        FuUnicodeCodepointCaseConvert := 66571;
        RETURN;
    66612:
        FuUnicodeCodepointCaseConvert := 66572;
        RETURN;
    66613:
        FuUnicodeCodepointCaseConvert := 66573;
        RETURN;
    66614:
        FuUnicodeCodepointCaseConvert := 66574;
        RETURN;
    66615:
        FuUnicodeCodepointCaseConvert := 66575;
        RETURN;
    66616:
        FuUnicodeCodepointCaseConvert := 66576;
        RETURN;
    66617:
        FuUnicodeCodepointCaseConvert := 66577;
        RETURN;
    66618:
        FuUnicodeCodepointCaseConvert := 66578;
        RETURN;
    66619:
        FuUnicodeCodepointCaseConvert := 66579;
        RETURN;
    66620:
        FuUnicodeCodepointCaseConvert := 66580;
        RETURN;
    66621:
        FuUnicodeCodepointCaseConvert := 66581;
        RETURN;
    66622:
        FuUnicodeCodepointCaseConvert := 66582;
        RETURN;
    66623:
        FuUnicodeCodepointCaseConvert := 66583;
        RETURN;
    66624:
        FuUnicodeCodepointCaseConvert := 66584;
        RETURN;
    66625:
        FuUnicodeCodepointCaseConvert := 66585;
        RETURN;
    66626:
        FuUnicodeCodepointCaseConvert := 66586;
        RETURN;
    66627:
        FuUnicodeCodepointCaseConvert := 66587;
        RETURN;
    66628:
        FuUnicodeCodepointCaseConvert := 66588;
        RETURN;
    66629:
        FuUnicodeCodepointCaseConvert := 66589;
        RETURN;
    66630:
        FuUnicodeCodepointCaseConvert := 66590;
        RETURN;
    66631:
        FuUnicodeCodepointCaseConvert := 66591;
        RETURN;
    66632:
        FuUnicodeCodepointCaseConvert := 66592;
        RETURN;
    66633:
        FuUnicodeCodepointCaseConvert := 66593;
        RETURN;
    66634:
        FuUnicodeCodepointCaseConvert := 66594;
        RETURN;
    66635:
        FuUnicodeCodepointCaseConvert := 66595;
        RETURN;
    66636:
        FuUnicodeCodepointCaseConvert := 66596;
        RETURN;
    66637:
        FuUnicodeCodepointCaseConvert := 66597;
        RETURN;
    66638:
        FuUnicodeCodepointCaseConvert := 66598;
        RETURN;
    66639:
        FuUnicodeCodepointCaseConvert := 66599;
        RETURN;
    66736:
        FuUnicodeCodepointCaseConvert := 66776;
        RETURN;
    66737:
        FuUnicodeCodepointCaseConvert := 66777;
        RETURN;
    66738:
        FuUnicodeCodepointCaseConvert := 66778;
        RETURN;
    66739:
        FuUnicodeCodepointCaseConvert := 66779;
        RETURN;
    66740:
        FuUnicodeCodepointCaseConvert := 66780;
        RETURN;
    66741:
        FuUnicodeCodepointCaseConvert := 66781;
        RETURN;
    66742:
        FuUnicodeCodepointCaseConvert := 66782;
        RETURN;
    66743:
        FuUnicodeCodepointCaseConvert := 66783;
        RETURN;
    66744:
        FuUnicodeCodepointCaseConvert := 66784;
        RETURN;
    66745:
        FuUnicodeCodepointCaseConvert := 66785;
        RETURN;
    66746:
        FuUnicodeCodepointCaseConvert := 66786;
        RETURN;
    66747:
        FuUnicodeCodepointCaseConvert := 66787;
        RETURN;
    66748:
        FuUnicodeCodepointCaseConvert := 66788;
        RETURN;
    66749:
        FuUnicodeCodepointCaseConvert := 66789;
        RETURN;
    66750:
        FuUnicodeCodepointCaseConvert := 66790;
        RETURN;
    66751:
        FuUnicodeCodepointCaseConvert := 66791;
        RETURN;
    66752:
        FuUnicodeCodepointCaseConvert := 66792;
        RETURN;
    66753:
        FuUnicodeCodepointCaseConvert := 66793;
        RETURN;
    66754:
        FuUnicodeCodepointCaseConvert := 66794;
        RETURN;
    66755:
        FuUnicodeCodepointCaseConvert := 66795;
        RETURN;
    66756:
        FuUnicodeCodepointCaseConvert := 66796;
        RETURN;
    66757:
        FuUnicodeCodepointCaseConvert := 66797;
        RETURN;
    66758:
        FuUnicodeCodepointCaseConvert := 66798;
        RETURN;
    66759:
        FuUnicodeCodepointCaseConvert := 66799;
        RETURN;
    66760:
        FuUnicodeCodepointCaseConvert := 66800;
        RETURN;
    66761:
        FuUnicodeCodepointCaseConvert := 66801;
        RETURN;
    66762:
        FuUnicodeCodepointCaseConvert := 66802;
        RETURN;
    66763:
        FuUnicodeCodepointCaseConvert := 66803;
        RETURN;
    66764:
        FuUnicodeCodepointCaseConvert := 66804;
        RETURN;
    66765:
        FuUnicodeCodepointCaseConvert := 66805;
        RETURN;
    66766:
        FuUnicodeCodepointCaseConvert := 66806;
        RETURN;
    66767:
        FuUnicodeCodepointCaseConvert := 66807;
        RETURN;
    66768:
        FuUnicodeCodepointCaseConvert := 66808;
        RETURN;
    66769:
        FuUnicodeCodepointCaseConvert := 66809;
        RETURN;
    66770:
        FuUnicodeCodepointCaseConvert := 66810;
        RETURN;
    66771:
        FuUnicodeCodepointCaseConvert := 66811;
        RETURN;
    66776:
        FuUnicodeCodepointCaseConvert := 66736;
        RETURN;
    66777:
        FuUnicodeCodepointCaseConvert := 66737;
        RETURN;
    66778:
        FuUnicodeCodepointCaseConvert := 66738;
        RETURN;
    66779:
        FuUnicodeCodepointCaseConvert := 66739;
        RETURN;
    66780:
        FuUnicodeCodepointCaseConvert := 66740;
        RETURN;
    66781:
        FuUnicodeCodepointCaseConvert := 66741;
        RETURN;
    66782:
        FuUnicodeCodepointCaseConvert := 66742;
        RETURN;
    66783:
        FuUnicodeCodepointCaseConvert := 66743;
        RETURN;
    66784:
        FuUnicodeCodepointCaseConvert := 66744;
        RETURN;
    66785:
        FuUnicodeCodepointCaseConvert := 66745;
        RETURN;
    66786:
        FuUnicodeCodepointCaseConvert := 66746;
        RETURN;
    66787:
        FuUnicodeCodepointCaseConvert := 66747;
        RETURN;
    66788:
        FuUnicodeCodepointCaseConvert := 66748;
        RETURN;
    66789:
        FuUnicodeCodepointCaseConvert := 66749;
        RETURN;
    66790:
        FuUnicodeCodepointCaseConvert := 66750;
        RETURN;
    66791:
        FuUnicodeCodepointCaseConvert := 66751;
        RETURN;
    66792:
        FuUnicodeCodepointCaseConvert := 66752;
        RETURN;
    66793:
        FuUnicodeCodepointCaseConvert := 66753;
        RETURN;
    66794:
        FuUnicodeCodepointCaseConvert := 66754;
        RETURN;
    66795:
        FuUnicodeCodepointCaseConvert := 66755;
        RETURN;
    66796:
        FuUnicodeCodepointCaseConvert := 66756;
        RETURN;
    66797:
        FuUnicodeCodepointCaseConvert := 66757;
        RETURN;
    66798:
        FuUnicodeCodepointCaseConvert := 66758;
        RETURN;
    66799:
        FuUnicodeCodepointCaseConvert := 66759;
        RETURN;
    66800:
        FuUnicodeCodepointCaseConvert := 66760;
        RETURN;
    66801:
        FuUnicodeCodepointCaseConvert := 66761;
        RETURN;
    66802:
        FuUnicodeCodepointCaseConvert := 66762;
        RETURN;
    66803:
        FuUnicodeCodepointCaseConvert := 66763;
        RETURN;
    66804:
        FuUnicodeCodepointCaseConvert := 66764;
        RETURN;
    66805:
        FuUnicodeCodepointCaseConvert := 66765;
        RETURN;
    66806:
        FuUnicodeCodepointCaseConvert := 66766;
        RETURN;
    66807:
        FuUnicodeCodepointCaseConvert := 66767;
        RETURN;
    66808:
        FuUnicodeCodepointCaseConvert := 66768;
        RETURN;
    66809:
        FuUnicodeCodepointCaseConvert := 66769;
        RETURN;
    66810:
        FuUnicodeCodepointCaseConvert := 66770;
        RETURN;
    66811:
        FuUnicodeCodepointCaseConvert := 66771;
        RETURN;
    66928:
        FuUnicodeCodepointCaseConvert := 66967;
        RETURN;
    66929:
        FuUnicodeCodepointCaseConvert := 66968;
        RETURN;
    66930:
        FuUnicodeCodepointCaseConvert := 66969;
        RETURN;
    66931:
        FuUnicodeCodepointCaseConvert := 66970;
        RETURN;
    66932:
        FuUnicodeCodepointCaseConvert := 66971;
        RETURN;
    66933:
        FuUnicodeCodepointCaseConvert := 66972;
        RETURN;
    66934:
        FuUnicodeCodepointCaseConvert := 66973;
        RETURN;
    66935:
        FuUnicodeCodepointCaseConvert := 66974;
        RETURN;
    66936:
        FuUnicodeCodepointCaseConvert := 66975;
        RETURN;
    66937:
        FuUnicodeCodepointCaseConvert := 66976;
        RETURN;
    66938:
        FuUnicodeCodepointCaseConvert := 66977;
        RETURN;
    66940:
        FuUnicodeCodepointCaseConvert := 66979;
        RETURN;
    66941:
        FuUnicodeCodepointCaseConvert := 66980;
        RETURN;
    66942:
        FuUnicodeCodepointCaseConvert := 66981;
        RETURN;
    66943:
        FuUnicodeCodepointCaseConvert := 66982;
        RETURN;
    66944:
        FuUnicodeCodepointCaseConvert := 66983;
        RETURN;
    66945:
        FuUnicodeCodepointCaseConvert := 66984;
        RETURN;
    66946:
        FuUnicodeCodepointCaseConvert := 66985;
        RETURN;
    66947:
        FuUnicodeCodepointCaseConvert := 66986;
        RETURN;
    66948:
        FuUnicodeCodepointCaseConvert := 66987;
        RETURN;
    66949:
        FuUnicodeCodepointCaseConvert := 66988;
        RETURN;
    66950:
        FuUnicodeCodepointCaseConvert := 66989;
        RETURN;
    66951:
        FuUnicodeCodepointCaseConvert := 66990;
        RETURN;
    66952:
        FuUnicodeCodepointCaseConvert := 66991;
        RETURN;
    66953:
        FuUnicodeCodepointCaseConvert := 66992;
        RETURN;
    66954:
        FuUnicodeCodepointCaseConvert := 66993;
        RETURN;
    66956:
        FuUnicodeCodepointCaseConvert := 66995;
        RETURN;
    66957:
        FuUnicodeCodepointCaseConvert := 66996;
        RETURN;
    66958:
        FuUnicodeCodepointCaseConvert := 66997;
        RETURN;
    66959:
        FuUnicodeCodepointCaseConvert := 66998;
        RETURN;
    66960:
        FuUnicodeCodepointCaseConvert := 66999;
        RETURN;
    66961:
        FuUnicodeCodepointCaseConvert := 67000;
        RETURN;
    66962:
        FuUnicodeCodepointCaseConvert := 67001;
        RETURN;
    66964:
        FuUnicodeCodepointCaseConvert := 67003;
        RETURN;
    66965:
        FuUnicodeCodepointCaseConvert := 67004;
        RETURN;
    66967:
        FuUnicodeCodepointCaseConvert := 66928;
        RETURN;
    66968:
        FuUnicodeCodepointCaseConvert := 66929;
        RETURN;
    66969:
        FuUnicodeCodepointCaseConvert := 66930;
        RETURN;
    66970:
        FuUnicodeCodepointCaseConvert := 66931;
        RETURN;
    66971:
        FuUnicodeCodepointCaseConvert := 66932;
        RETURN;
    66972:
        FuUnicodeCodepointCaseConvert := 66933;
        RETURN;
    66973:
        FuUnicodeCodepointCaseConvert := 66934;
        RETURN;
    66974:
        FuUnicodeCodepointCaseConvert := 66935;
        RETURN;
    66975:
        FuUnicodeCodepointCaseConvert := 66936;
        RETURN;
    66976:
        FuUnicodeCodepointCaseConvert := 66937;
        RETURN;
    66977:
        FuUnicodeCodepointCaseConvert := 66938;
        RETURN;
    66979:
        FuUnicodeCodepointCaseConvert := 66940;
        RETURN;
    66980:
        FuUnicodeCodepointCaseConvert := 66941;
        RETURN;
    66981:
        FuUnicodeCodepointCaseConvert := 66942;
        RETURN;
    66982:
        FuUnicodeCodepointCaseConvert := 66943;
        RETURN;
    66983:
        FuUnicodeCodepointCaseConvert := 66944;
        RETURN;
    66984:
        FuUnicodeCodepointCaseConvert := 66945;
        RETURN;
    66985:
        FuUnicodeCodepointCaseConvert := 66946;
        RETURN;
    66986:
        FuUnicodeCodepointCaseConvert := 66947;
        RETURN;
    66987:
        FuUnicodeCodepointCaseConvert := 66948;
        RETURN;
    66988:
        FuUnicodeCodepointCaseConvert := 66949;
        RETURN;
    66989:
        FuUnicodeCodepointCaseConvert := 66950;
        RETURN;
    66990:
        FuUnicodeCodepointCaseConvert := 66951;
        RETURN;
    66991:
        FuUnicodeCodepointCaseConvert := 66952;
        RETURN;
    66992:
        FuUnicodeCodepointCaseConvert := 66953;
        RETURN;
    66993:
        FuUnicodeCodepointCaseConvert := 66954;
        RETURN;
    66995:
        FuUnicodeCodepointCaseConvert := 66956;
        RETURN;
    66996:
        FuUnicodeCodepointCaseConvert := 66957;
        RETURN;
    66997:
        FuUnicodeCodepointCaseConvert := 66958;
        RETURN;
    66998:
        FuUnicodeCodepointCaseConvert := 66959;
        RETURN;
    66999:
        FuUnicodeCodepointCaseConvert := 66960;
        RETURN;
    67000:
        FuUnicodeCodepointCaseConvert := 66961;
        RETURN;
    67001:
        FuUnicodeCodepointCaseConvert := 66962;
        RETURN;
    67003:
        FuUnicodeCodepointCaseConvert := 66964;
        RETURN;
    67004:
        FuUnicodeCodepointCaseConvert := 66965;
        RETURN;
    68736:
        FuUnicodeCodepointCaseConvert := 68800;
        RETURN;
    68737:
        FuUnicodeCodepointCaseConvert := 68801;
        RETURN;
    68738:
        FuUnicodeCodepointCaseConvert := 68802;
        RETURN;
    68739:
        FuUnicodeCodepointCaseConvert := 68803;
        RETURN;
    68740:
        FuUnicodeCodepointCaseConvert := 68804;
        RETURN;
    68741:
        FuUnicodeCodepointCaseConvert := 68805;
        RETURN;
    68742:
        FuUnicodeCodepointCaseConvert := 68806;
        RETURN;
    68743:
        FuUnicodeCodepointCaseConvert := 68807;
        RETURN;
    68744:
        FuUnicodeCodepointCaseConvert := 68808;
        RETURN;
    68745:
        FuUnicodeCodepointCaseConvert := 68809;
        RETURN;
    68746:
        FuUnicodeCodepointCaseConvert := 68810;
        RETURN;
    68747:
        FuUnicodeCodepointCaseConvert := 68811;
        RETURN;
    68748:
        FuUnicodeCodepointCaseConvert := 68812;
        RETURN;
    68749:
        FuUnicodeCodepointCaseConvert := 68813;
        RETURN;
    68750:
        FuUnicodeCodepointCaseConvert := 68814;
        RETURN;
    68751:
        FuUnicodeCodepointCaseConvert := 68815;
        RETURN;
    68752:
        FuUnicodeCodepointCaseConvert := 68816;
        RETURN;
    68753:
        FuUnicodeCodepointCaseConvert := 68817;
        RETURN;
    68754:
        FuUnicodeCodepointCaseConvert := 68818;
        RETURN;
    68755:
        FuUnicodeCodepointCaseConvert := 68819;
        RETURN;
    68756:
        FuUnicodeCodepointCaseConvert := 68820;
        RETURN;
    68757:
        FuUnicodeCodepointCaseConvert := 68821;
        RETURN;
    68758:
        FuUnicodeCodepointCaseConvert := 68822;
        RETURN;
    68759:
        FuUnicodeCodepointCaseConvert := 68823;
        RETURN;
    68760:
        FuUnicodeCodepointCaseConvert := 68824;
        RETURN;
    68761:
        FuUnicodeCodepointCaseConvert := 68825;
        RETURN;
    68762:
        FuUnicodeCodepointCaseConvert := 68826;
        RETURN;
    68763:
        FuUnicodeCodepointCaseConvert := 68827;
        RETURN;
    68764:
        FuUnicodeCodepointCaseConvert := 68828;
        RETURN;
    68765:
        FuUnicodeCodepointCaseConvert := 68829;
        RETURN;
    68766:
        FuUnicodeCodepointCaseConvert := 68830;
        RETURN;
    68767:
        FuUnicodeCodepointCaseConvert := 68831;
        RETURN;
    68768:
        FuUnicodeCodepointCaseConvert := 68832;
        RETURN;
    68769:
        FuUnicodeCodepointCaseConvert := 68833;
        RETURN;
    68770:
        FuUnicodeCodepointCaseConvert := 68834;
        RETURN;
    68771:
        FuUnicodeCodepointCaseConvert := 68835;
        RETURN;
    68772:
        FuUnicodeCodepointCaseConvert := 68836;
        RETURN;
    68773:
        FuUnicodeCodepointCaseConvert := 68837;
        RETURN;
    68774:
        FuUnicodeCodepointCaseConvert := 68838;
        RETURN;
    68775:
        FuUnicodeCodepointCaseConvert := 68839;
        RETURN;
    68776:
        FuUnicodeCodepointCaseConvert := 68840;
        RETURN;
    68777:
        FuUnicodeCodepointCaseConvert := 68841;
        RETURN;
    68778:
        FuUnicodeCodepointCaseConvert := 68842;
        RETURN;
    68779:
        FuUnicodeCodepointCaseConvert := 68843;
        RETURN;
    68780:
        FuUnicodeCodepointCaseConvert := 68844;
        RETURN;
    68781:
        FuUnicodeCodepointCaseConvert := 68845;
        RETURN;
    68782:
        FuUnicodeCodepointCaseConvert := 68846;
        RETURN;
    68783:
        FuUnicodeCodepointCaseConvert := 68847;
        RETURN;
    68784:
        FuUnicodeCodepointCaseConvert := 68848;
        RETURN;
    68785:
        FuUnicodeCodepointCaseConvert := 68849;
        RETURN;
    68786:
        FuUnicodeCodepointCaseConvert := 68850;
        RETURN;
    68800:
        FuUnicodeCodepointCaseConvert := 68736;
        RETURN;
    68801:
        FuUnicodeCodepointCaseConvert := 68737;
        RETURN;
    68802:
        FuUnicodeCodepointCaseConvert := 68738;
        RETURN;
    68803:
        FuUnicodeCodepointCaseConvert := 68739;
        RETURN;
    68804:
        FuUnicodeCodepointCaseConvert := 68740;
        RETURN;
    68805:
        FuUnicodeCodepointCaseConvert := 68741;
        RETURN;
    68806:
        FuUnicodeCodepointCaseConvert := 68742;
        RETURN;
    68807:
        FuUnicodeCodepointCaseConvert := 68743;
        RETURN;
    68808:
        FuUnicodeCodepointCaseConvert := 68744;
        RETURN;
    68809:
        FuUnicodeCodepointCaseConvert := 68745;
        RETURN;
    68810:
        FuUnicodeCodepointCaseConvert := 68746;
        RETURN;
    68811:
        FuUnicodeCodepointCaseConvert := 68747;
        RETURN;
    68812:
        FuUnicodeCodepointCaseConvert := 68748;
        RETURN;
    68813:
        FuUnicodeCodepointCaseConvert := 68749;
        RETURN;
    68814:
        FuUnicodeCodepointCaseConvert := 68750;
        RETURN;
    68815:
        FuUnicodeCodepointCaseConvert := 68751;
        RETURN;
    68816:
        FuUnicodeCodepointCaseConvert := 68752;
        RETURN;
    68817:
        FuUnicodeCodepointCaseConvert := 68753;
        RETURN;
    68818:
        FuUnicodeCodepointCaseConvert := 68754;
        RETURN;
    68819:
        FuUnicodeCodepointCaseConvert := 68755;
        RETURN;
    68820:
        FuUnicodeCodepointCaseConvert := 68756;
        RETURN;
    68821:
        FuUnicodeCodepointCaseConvert := 68757;
        RETURN;
    68822:
        FuUnicodeCodepointCaseConvert := 68758;
        RETURN;
    68823:
        FuUnicodeCodepointCaseConvert := 68759;
        RETURN;
    68824:
        FuUnicodeCodepointCaseConvert := 68760;
        RETURN;
    68825:
        FuUnicodeCodepointCaseConvert := 68761;
        RETURN;
    68826:
        FuUnicodeCodepointCaseConvert := 68762;
        RETURN;
    68827:
        FuUnicodeCodepointCaseConvert := 68763;
        RETURN;
    68828:
        FuUnicodeCodepointCaseConvert := 68764;
        RETURN;
    68829:
        FuUnicodeCodepointCaseConvert := 68765;
        RETURN;
    68830:
        FuUnicodeCodepointCaseConvert := 68766;
        RETURN;
    68831:
        FuUnicodeCodepointCaseConvert := 68767;
        RETURN;
    68832:
        FuUnicodeCodepointCaseConvert := 68768;
        RETURN;
    68833:
        FuUnicodeCodepointCaseConvert := 68769;
        RETURN;
    68834:
        FuUnicodeCodepointCaseConvert := 68770;
        RETURN;
    68835:
        FuUnicodeCodepointCaseConvert := 68771;
        RETURN;
    68836:
        FuUnicodeCodepointCaseConvert := 68772;
        RETURN;
    68837:
        FuUnicodeCodepointCaseConvert := 68773;
        RETURN;
    68838:
        FuUnicodeCodepointCaseConvert := 68774;
        RETURN;
    68839:
        FuUnicodeCodepointCaseConvert := 68775;
        RETURN;
    68840:
        FuUnicodeCodepointCaseConvert := 68776;
        RETURN;
    68841:
        FuUnicodeCodepointCaseConvert := 68777;
        RETURN;
    68842:
        FuUnicodeCodepointCaseConvert := 68778;
        RETURN;
    68843:
        FuUnicodeCodepointCaseConvert := 68779;
        RETURN;
    68844:
        FuUnicodeCodepointCaseConvert := 68780;
        RETURN;
    68845:
        FuUnicodeCodepointCaseConvert := 68781;
        RETURN;
    68846:
        FuUnicodeCodepointCaseConvert := 68782;
        RETURN;
    68847:
        FuUnicodeCodepointCaseConvert := 68783;
        RETURN;
    68848:
        FuUnicodeCodepointCaseConvert := 68784;
        RETURN;
    68849:
        FuUnicodeCodepointCaseConvert := 68785;
        RETURN;
    68850:
        FuUnicodeCodepointCaseConvert := 68786;
        RETURN;
    71840:
        FuUnicodeCodepointCaseConvert := 71872;
        RETURN;
    71841:
        FuUnicodeCodepointCaseConvert := 71873;
        RETURN;
    71842:
        FuUnicodeCodepointCaseConvert := 71874;
        RETURN;
    71843:
        FuUnicodeCodepointCaseConvert := 71875;
        RETURN;
    71844:
        FuUnicodeCodepointCaseConvert := 71876;
        RETURN;
    71845:
        FuUnicodeCodepointCaseConvert := 71877;
        RETURN;
    71846:
        FuUnicodeCodepointCaseConvert := 71878;
        RETURN;
    71847:
        FuUnicodeCodepointCaseConvert := 71879;
        RETURN;
    71848:
        FuUnicodeCodepointCaseConvert := 71880;
        RETURN;
    71849:
        FuUnicodeCodepointCaseConvert := 71881;
        RETURN;
    71850:
        FuUnicodeCodepointCaseConvert := 71882;
        RETURN;
    71851:
        FuUnicodeCodepointCaseConvert := 71883;
        RETURN;
    71852:
        FuUnicodeCodepointCaseConvert := 71884;
        RETURN;
    71853:
        FuUnicodeCodepointCaseConvert := 71885;
        RETURN;
    71854:
        FuUnicodeCodepointCaseConvert := 71886;
        RETURN;
    71855:
        FuUnicodeCodepointCaseConvert := 71887;
        RETURN;
    71856:
        FuUnicodeCodepointCaseConvert := 71888;
        RETURN;
    71857:
        FuUnicodeCodepointCaseConvert := 71889;
        RETURN;
    71858:
        FuUnicodeCodepointCaseConvert := 71890;
        RETURN;
    71859:
        FuUnicodeCodepointCaseConvert := 71891;
        RETURN;
    71860:
        FuUnicodeCodepointCaseConvert := 71892;
        RETURN;
    71861:
        FuUnicodeCodepointCaseConvert := 71893;
        RETURN;
    71862:
        FuUnicodeCodepointCaseConvert := 71894;
        RETURN;
    71863:
        FuUnicodeCodepointCaseConvert := 71895;
        RETURN;
    71864:
        FuUnicodeCodepointCaseConvert := 71896;
        RETURN;
    71865:
        FuUnicodeCodepointCaseConvert := 71897;
        RETURN;
    71866:
        FuUnicodeCodepointCaseConvert := 71898;
        RETURN;
    71867:
        FuUnicodeCodepointCaseConvert := 71899;
        RETURN;
    71868:
        FuUnicodeCodepointCaseConvert := 71900;
        RETURN;
    71869:
        FuUnicodeCodepointCaseConvert := 71901;
        RETURN;
    71870:
        FuUnicodeCodepointCaseConvert := 71902;
        RETURN;
    71871:
        FuUnicodeCodepointCaseConvert := 71903;
        RETURN;
    71872:
        FuUnicodeCodepointCaseConvert := 71840;
        RETURN;
    71873:
        FuUnicodeCodepointCaseConvert := 71841;
        RETURN;
    71874:
        FuUnicodeCodepointCaseConvert := 71842;
        RETURN;
    71875:
        FuUnicodeCodepointCaseConvert := 71843;
        RETURN;
    71876:
        FuUnicodeCodepointCaseConvert := 71844;
        RETURN;
    71877:
        FuUnicodeCodepointCaseConvert := 71845;
        RETURN;
    71878:
        FuUnicodeCodepointCaseConvert := 71846;
        RETURN;
    71879:
        FuUnicodeCodepointCaseConvert := 71847;
        RETURN;
    71880:
        FuUnicodeCodepointCaseConvert := 71848;
        RETURN;
    71881:
        FuUnicodeCodepointCaseConvert := 71849;
        RETURN;
    71882:
        FuUnicodeCodepointCaseConvert := 71850;
        RETURN;
    71883:
        FuUnicodeCodepointCaseConvert := 71851;
        RETURN;
    71884:
        FuUnicodeCodepointCaseConvert := 71852;
        RETURN;
    71885:
        FuUnicodeCodepointCaseConvert := 71853;
        RETURN;
    71886:
        FuUnicodeCodepointCaseConvert := 71854;
        RETURN;
    71887:
        FuUnicodeCodepointCaseConvert := 71855;
        RETURN;
    71888:
        FuUnicodeCodepointCaseConvert := 71856;
        RETURN;
    71889:
        FuUnicodeCodepointCaseConvert := 71857;
        RETURN;
    71890:
        FuUnicodeCodepointCaseConvert := 71858;
        RETURN;
    71891:
        FuUnicodeCodepointCaseConvert := 71859;
        RETURN;
    71892:
        FuUnicodeCodepointCaseConvert := 71860;
        RETURN;
    71893:
        FuUnicodeCodepointCaseConvert := 71861;
        RETURN;
    71894:
        FuUnicodeCodepointCaseConvert := 71862;
        RETURN;
    71895:
        FuUnicodeCodepointCaseConvert := 71863;
        RETURN;
    71896:
        FuUnicodeCodepointCaseConvert := 71864;
        RETURN;
    71897:
        FuUnicodeCodepointCaseConvert := 71865;
        RETURN;
    71898:
        FuUnicodeCodepointCaseConvert := 71866;
        RETURN;
    71899:
        FuUnicodeCodepointCaseConvert := 71867;
        RETURN;
    71900:
        FuUnicodeCodepointCaseConvert := 71868;
        RETURN;
    71901:
        FuUnicodeCodepointCaseConvert := 71869;
        RETURN;
    71902:
        FuUnicodeCodepointCaseConvert := 71870;
        RETURN;
    71903:
        FuUnicodeCodepointCaseConvert := 71871;
        RETURN;
    93760:
        FuUnicodeCodepointCaseConvert := 93792;
        RETURN;
    93761:
        FuUnicodeCodepointCaseConvert := 93793;
        RETURN;
    93762:
        FuUnicodeCodepointCaseConvert := 93794;
        RETURN;
    93763:
        FuUnicodeCodepointCaseConvert := 93795;
        RETURN;
    93764:
        FuUnicodeCodepointCaseConvert := 93796;
        RETURN;
    93765:
        FuUnicodeCodepointCaseConvert := 93797;
        RETURN;
    93766:
        FuUnicodeCodepointCaseConvert := 93798;
        RETURN;
    93767:
        FuUnicodeCodepointCaseConvert := 93799;
        RETURN;
    93768:
        FuUnicodeCodepointCaseConvert := 93800;
        RETURN;
    93769:
        FuUnicodeCodepointCaseConvert := 93801;
        RETURN;
    93770:
        FuUnicodeCodepointCaseConvert := 93802;
        RETURN;
    93771:
        FuUnicodeCodepointCaseConvert := 93803;
        RETURN;
    93772:
        FuUnicodeCodepointCaseConvert := 93804;
        RETURN;
    93773:
        FuUnicodeCodepointCaseConvert := 93805;
        RETURN;
    93774:
        FuUnicodeCodepointCaseConvert := 93806;
        RETURN;
    93775:
        FuUnicodeCodepointCaseConvert := 93807;
        RETURN;
    93776:
        FuUnicodeCodepointCaseConvert := 93808;
        RETURN;
    93777:
        FuUnicodeCodepointCaseConvert := 93809;
        RETURN;
    93778:
        FuUnicodeCodepointCaseConvert := 93810;
        RETURN;
    93779:
        FuUnicodeCodepointCaseConvert := 93811;
        RETURN;
    93780:
        FuUnicodeCodepointCaseConvert := 93812;
        RETURN;
    93781:
        FuUnicodeCodepointCaseConvert := 93813;
        RETURN;
    93782:
        FuUnicodeCodepointCaseConvert := 93814;
        RETURN;
    93783:
        FuUnicodeCodepointCaseConvert := 93815;
        RETURN;
    93784:
        FuUnicodeCodepointCaseConvert := 93816;
        RETURN;
    93785:
        FuUnicodeCodepointCaseConvert := 93817;
        RETURN;
    93786:
        FuUnicodeCodepointCaseConvert := 93818;
        RETURN;
    93787:
        FuUnicodeCodepointCaseConvert := 93819;
        RETURN;
    93788:
        FuUnicodeCodepointCaseConvert := 93820;
        RETURN;
    93789:
        FuUnicodeCodepointCaseConvert := 93821;
        RETURN;
    93790:
        FuUnicodeCodepointCaseConvert := 93822;
        RETURN;
    93791:
        FuUnicodeCodepointCaseConvert := 93823;
        RETURN;
    93792:
        FuUnicodeCodepointCaseConvert := 93760;
        RETURN;
    93793:
        FuUnicodeCodepointCaseConvert := 93761;
        RETURN;
    93794:
        FuUnicodeCodepointCaseConvert := 93762;
        RETURN;
    93795:
        FuUnicodeCodepointCaseConvert := 93763;
        RETURN;
    93796:
        FuUnicodeCodepointCaseConvert := 93764;
        RETURN;
    93797:
        FuUnicodeCodepointCaseConvert := 93765;
        RETURN;
    93798:
        FuUnicodeCodepointCaseConvert := 93766;
        RETURN;
    93799:
        FuUnicodeCodepointCaseConvert := 93767;
        RETURN;
    93800:
        FuUnicodeCodepointCaseConvert := 93768;
        RETURN;
    93801:
        FuUnicodeCodepointCaseConvert := 93769;
        RETURN;
    93802:
        FuUnicodeCodepointCaseConvert := 93770;
        RETURN;
    93803:
        FuUnicodeCodepointCaseConvert := 93771;
        RETURN;
    93804:
        FuUnicodeCodepointCaseConvert := 93772;
        RETURN;
    93805:
        FuUnicodeCodepointCaseConvert := 93773;
        RETURN;
    93806:
        FuUnicodeCodepointCaseConvert := 93774;
        RETURN;
    93807:
        FuUnicodeCodepointCaseConvert := 93775;
        RETURN;
    93808:
        FuUnicodeCodepointCaseConvert := 93776;
        RETURN;
    93809:
        FuUnicodeCodepointCaseConvert := 93777;
        RETURN;
    93810:
        FuUnicodeCodepointCaseConvert := 93778;
        RETURN;
    93811:
        FuUnicodeCodepointCaseConvert := 93779;
        RETURN;
    93812:
        FuUnicodeCodepointCaseConvert := 93780;
        RETURN;
    93813:
        FuUnicodeCodepointCaseConvert := 93781;
        RETURN;
    93814:
        FuUnicodeCodepointCaseConvert := 93782;
        RETURN;
    93815:
        FuUnicodeCodepointCaseConvert := 93783;
        RETURN;
    93816:
        FuUnicodeCodepointCaseConvert := 93784;
        RETURN;
    93817:
        FuUnicodeCodepointCaseConvert := 93785;
        RETURN;
    93818:
        FuUnicodeCodepointCaseConvert := 93786;
        RETURN;
    93819:
        FuUnicodeCodepointCaseConvert := 93787;
        RETURN;
    93820:
        FuUnicodeCodepointCaseConvert := 93788;
        RETURN;
    93821:
        FuUnicodeCodepointCaseConvert := 93789;
        RETURN;
    93822:
        FuUnicodeCodepointCaseConvert := 93790;
        RETURN;
    93823:
        FuUnicodeCodepointCaseConvert := 93791;
        RETURN;
    125184:
        FuUnicodeCodepointCaseConvert := 125218;
        RETURN;
    125185:
        FuUnicodeCodepointCaseConvert := 125219;
        RETURN;
    125186:
        FuUnicodeCodepointCaseConvert := 125220;
        RETURN;
    125187:
        FuUnicodeCodepointCaseConvert := 125221;
        RETURN;
    125188:
        FuUnicodeCodepointCaseConvert := 125222;
        RETURN;
    125189:
        FuUnicodeCodepointCaseConvert := 125223;
        RETURN;
    125190:
        FuUnicodeCodepointCaseConvert := 125224;
        RETURN;
    125191:
        FuUnicodeCodepointCaseConvert := 125225;
        RETURN;
    125192:
        FuUnicodeCodepointCaseConvert := 125226;
        RETURN;
    125193:
        FuUnicodeCodepointCaseConvert := 125227;
        RETURN;
    125194:
        FuUnicodeCodepointCaseConvert := 125228;
        RETURN;
    125195:
        FuUnicodeCodepointCaseConvert := 125229;
        RETURN;
    125196:
        FuUnicodeCodepointCaseConvert := 125230;
        RETURN;
    125197:
        FuUnicodeCodepointCaseConvert := 125231;
        RETURN;
    125198:
        FuUnicodeCodepointCaseConvert := 125232;
        RETURN;
    125199:
        FuUnicodeCodepointCaseConvert := 125233;
        RETURN;
    125200:
        FuUnicodeCodepointCaseConvert := 125234;
        RETURN;
    125201:
        FuUnicodeCodepointCaseConvert := 125235;
        RETURN;
    125202:
        FuUnicodeCodepointCaseConvert := 125236;
        RETURN;
    125203:
        FuUnicodeCodepointCaseConvert := 125237;
        RETURN;
    125204:
        FuUnicodeCodepointCaseConvert := 125238;
        RETURN;
    125205:
        FuUnicodeCodepointCaseConvert := 125239;
        RETURN;
    125206:
        FuUnicodeCodepointCaseConvert := 125240;
        RETURN;
    125207:
        FuUnicodeCodepointCaseConvert := 125241;
        RETURN;
    125208:
        FuUnicodeCodepointCaseConvert := 125242;
        RETURN;
    125209:
        FuUnicodeCodepointCaseConvert := 125243;
        RETURN;
    125210:
        FuUnicodeCodepointCaseConvert := 125244;
        RETURN;
    125211:
        FuUnicodeCodepointCaseConvert := 125245;
        RETURN;
    125212:
        FuUnicodeCodepointCaseConvert := 125246;
        RETURN;
    125213:
        FuUnicodeCodepointCaseConvert := 125247;
        RETURN;
    125214:
        FuUnicodeCodepointCaseConvert := 125248;
        RETURN;
    125215:
        FuUnicodeCodepointCaseConvert := 125249;
        RETURN;
    125216:
        FuUnicodeCodepointCaseConvert := 125250;
        RETURN;
    125217:
        FuUnicodeCodepointCaseConvert := 125251;
        RETURN;
    125218:
        FuUnicodeCodepointCaseConvert := 125184;
        RETURN;
    125219:
        FuUnicodeCodepointCaseConvert := 125185;
        RETURN;
    125220:
        FuUnicodeCodepointCaseConvert := 125186;
        RETURN;
    125221:
        FuUnicodeCodepointCaseConvert := 125187;
        RETURN;
    125222:
        FuUnicodeCodepointCaseConvert := 125188;
        RETURN;
    125223:
        FuUnicodeCodepointCaseConvert := 125189;
        RETURN;
    125224:
        FuUnicodeCodepointCaseConvert := 125190;
        RETURN;
    125225:
        FuUnicodeCodepointCaseConvert := 125191;
        RETURN;
    125226:
        FuUnicodeCodepointCaseConvert := 125192;
        RETURN;
    125227:
        FuUnicodeCodepointCaseConvert := 125193;
        RETURN;
    125228:
        FuUnicodeCodepointCaseConvert := 125194;
        RETURN;
    125229:
        FuUnicodeCodepointCaseConvert := 125195;
        RETURN;
    125230:
        FuUnicodeCodepointCaseConvert := 125196;
        RETURN;
    125231:
        FuUnicodeCodepointCaseConvert := 125197;
        RETURN;
    125232:
        FuUnicodeCodepointCaseConvert := 125198;
        RETURN;
    125233:
        FuUnicodeCodepointCaseConvert := 125199;
        RETURN;
    125234:
        FuUnicodeCodepointCaseConvert := 125200;
        RETURN;
    125235:
        FuUnicodeCodepointCaseConvert := 125201;
        RETURN;
    125236:
        FuUnicodeCodepointCaseConvert := 125202;
        RETURN;
    125237:
        FuUnicodeCodepointCaseConvert := 125203;
        RETURN;
    125238:
        FuUnicodeCodepointCaseConvert := 125204;
        RETURN;
    125239:
        FuUnicodeCodepointCaseConvert := 125205;
        RETURN;
    125240:
        FuUnicodeCodepointCaseConvert := 125206;
        RETURN;
    125241:
        FuUnicodeCodepointCaseConvert := 125207;
        RETURN;
    125242:
        FuUnicodeCodepointCaseConvert := 125208;
        RETURN;
    125243:
        FuUnicodeCodepointCaseConvert := 125209;
        RETURN;
    125244:
        FuUnicodeCodepointCaseConvert := 125210;
        RETURN;
    125245:
        FuUnicodeCodepointCaseConvert := 125211;
        RETURN;
    125246:
        FuUnicodeCodepointCaseConvert := 125212;
        RETURN;
    125247:
        FuUnicodeCodepointCaseConvert := 125213;
        RETURN;
    125248:
        FuUnicodeCodepointCaseConvert := 125214;
        RETURN;
    125249:
        FuUnicodeCodepointCaseConvert := 125215;
        RETURN;
    125250:
        FuUnicodeCodepointCaseConvert := 125216;
        RETURN;
    125251:
        FuUnicodeCodepointCaseConvert := 125217;
        RETURN;
END_CASE

END_FUNCTION

// 20 Program Organization Units/FuMatchExpressionUTF8
// Matches the given compiled pattern against the subject.
// This is the UTF-8 version of FuMatchExpression.
// Disabling strict conformity allows the usage of the extended ASCII alphabet (ISO 8859-1, decimal 160-255),
// as long as it doesn't form a valid UTF-8 byte sequence.
{attribute 'qualified_only'}
FUNCTION FuMatchExpressionUTF8 : BOOL
VAR_INPUT
    typPattern: typCompiledPatternW;      // The compiled pattern from "FuCompilePatternW"
    psSubject: POINTER TO STRING(1);      // A pointer to the subject string - for technical reasons this is a STRING(1), although any size is supported
    udiLength: UDINT;                     // The length of the subject string (in bytes, not codepoints)
    xStrictConformity: BOOL := TRUE;      // Require strict conformity to the Unicode standard
END_VAR
{library PRIVATE}
VAR
    tempPtrStr: POINTER TO BYTE;
    tempPtrStrMatching: POINTER TO BYTE;
    tempStrIndex: UDINT;
    tempStrIndexMatching: UDINT;
    
    i: UINT;
    j: UINT;
    k: LINT;
    
    tempChar: DWORD;
    tempCharLength: USINT;
    
    tempNextChar: DWORD;
    tempNextCharLength: DWORD;
    
    tempLaziness: BOOL;
    tempHasEndChar: BOOL;
    tempEndChar: DWORD;
    tempEndChar2: DWORD;
    
    tempWildcardSearchStart: LINT;
    tempWildcardSearchEnd: LINT;
    tempWildcardSearchBy: LINT;
    tempWildcardSearchOffset: UDINT;
    tempWildcardSearchSuccess: BOOL;
END_VAR

FuMatchExpressionUTF8 := FALSE;

IF typPattern.uiCountTokens = 0 OR_ELSE udiLength = 0 THEN
    RETURN;
END_IF

tempPtrStr := psSubject;
tempStrIndex := 0;

WHILE i < typPattern.uiCountTokens DO
    IF tempStrIndex >= udiLength THEN
        // Only if all following tokens are of type WILDCARD, we can allow a match to be positive
        FOR j := i TO (typPattern.uiCountTokens - 1) BY 1 DO
            IF typPattern.atTokens[j].eType <> eTokenType.WILDCARD THEN
                FuMatchExpressionUTF8 := FALSE;
                RETURN;
            END_IF
        END_FOR
        
        FuMatchExpressionUTF8 := TRUE;
        RETURN;
    END_IF
    
    IF
        NOT FuUtf8CharToDword(
            psInput := (tempPtrStr + tempStrIndex),
            udiStringLength := (udiLength - tempStrIndex),
            xStrictConformity := xStrictConformity,
            dwCodepoint => tempChar,
            usiByteLength => tempCharLength
        )
    THEN
        RETURN;
    END_IF
    
    CASE typPattern.atTokens[i].eType OF
        eTokenType.INVALID: // We shouldn't ever get an invalid token inside our token array that isn't behind our count
            RETURN;
        
        eTokenType.LITERAL:
            IF
                tempChar <> typPattern.atTokens[i].dwChar AND_THEN
                (
                    NOT typPattern.xCaseInsensitive OR_ELSE
                    typPattern.atTokens[i].dwAlternativeChar = 0 OR_ELSE
                    tempChar <> typPattern.atTokens[i].dwAlternativeChar
                ) 
            THEN
                RETURN;
            END_IF
            
            tempStrIndex := tempStrIndex + tempCharLength;
        
        eTokenType.ANYCHAR:
            tempStrIndex := tempStrIndex + tempCharLength;
        
        eTokenType.WILDCARD:
            tempLaziness := (typPattern.atTokens[i].dwChar = 1);
            tempHasEndChar := FALSE;
            
            FOR j := i + 1 TO (typPattern.uiCountTokens - 1) BY 1 DO
                IF typPattern.atTokens[j].eType = eTokenType.LITERAL THEN
                    tempHasEndChar := TRUE;
                    tempEndChar := typPattern.atTokens[j].dwChar;
                    tempEndChar2 := typPattern.atTokens[j].dwAlternativeChar;
                    EXIT;
                END_IF
            END_FOR
            
            // If we don't have any characters to match on at the end of the pattern, we match immediately
            IF NOT tempHasEndChar THEN
                FuMatchExpressionUTF8 := TRUE;
                RETURN;
            END_IF
            
            IF tempLaziness THEN
                // Advance token pointer once more because the next token is the laziness token we already used
                i := i + 1;
                
                // If the wildcard is lazy, search from front to back
                tempWildcardSearchStart := TO_LINT(tempStrIndex);
                tempWildcardSearchEnd := TO_LINT(udiLength);
                tempWildcardSearchBy := 1;
            ELSE
                // If the wildcard is NOT lazy, search from back to front (greedy!)
                tempWildcardSearchStart := TO_LINT(udiLength);
                tempWildcardSearchEnd := TO_LINT(tempStrIndex);
                tempWildcardSearchBy := -1;
            END_IF
            
            tempWildcardSearchSuccess := FALSE;
            tempWildcardSearchOffset := 0;
            
            FOR k := tempWildcardSearchStart TO tempWildcardSearchEnd BY tempWildcardSearchBy DO
                IF
                    FuUtf8CharToDword(
                        psInput := (tempPtrStr + LINT_TO___XWORD(k)),
                        udiStringLength := (udiLength - tempWildcardSearchOffset),
                        xStrictConformity := xStrictConformity,
                        dwCodepoint => tempNextChar,
                        usiByteLength => tempNextCharLength
                    )
                THEN
                    tempWildcardSearchOffset := tempWildcardSearchOffset + tempNextCharLength;
                    
                    IF
                        tempNextChar = tempEndChar OR_ELSE
                        (typPattern.xCaseInsensitive AND_THEN tempEndChar2 <> 0 AND_THEN tempNextChar = tempEndChar2)
                    THEN
                        tempWildcardSearchSuccess := TRUE;
                        tempStrIndex := TO_UDINT(k);
                        EXIT;
                    END_IF
                ELSE
                    tempWildcardSearchOffset := tempWildcardSearchOffset + 1;
                END_IF
            END_FOR
            
            IF NOT tempWildcardSearchSuccess THEN
                RETURN;
            END_IF
    END_CASE
    
    i := i + 1;
END_WHILE

FuMatchExpressionUTF8 := (tempStrIndex >= udiLength);

END_FUNCTION

// 20 Program Organization Units/FuCompilePatternW
// Compiles the pattern into a stream of tokens for matching.
// This is the UTF-16 (WSTRING) version of FuCompilePattern.
//
// The alphabet can be matched case insensitive,
// otherwise by default the pattern is case sensitive.
// The case mapping table is NOT completely covered,
// as such you MAY encounter missing case conversion
// for some languages.
//
// A few examples of valid patterns:
//  - 'A*bEd'
//  - 'A*?bEd'
//  - 'A.b*e*'
//  - '*A\.b\*e*'
//  - 'A?\bed'
//
// The return value signifies whether compilation was successful,
// or the given pattern is invalid.
{attribute 'qualified_only'}
FUNCTION FuCompilePatternW : BOOL
VAR_INPUT
    pwsPattern: POINTER TO WSTRING(1);    // The pattern string to compile - for technical reasons this is a WSTRING(1), although any length is supported
    udiPatternLength: UDINT;              // Pattern string length (in words (length in bytes/2), not codepoints)
    xCaseInsensitive: BOOL := FALSE;      // Whether the pattern is case insensitive
END_VAR
VAR_OUTPUT
    typPattern: typCompiledPatternW;      // The compiled pattern, for "FuMatchExpressionW"
END_VAR
{library PRIVATE}
VAR
    tempPointer: POINTER TO WSTRING(1);
    
    i: UDINT;
    
    tempChar: DWORD;
    tempCharLength: UDINT;
    
    tempNextChar: DWORD;
    tempNextCharLength: UDINT;
    
    tempIndex: UINT;
    tempMaxStrIndex: UDINT;
END_VAR
VAR CONSTANT
    CHAR_WILDCARD: DWORD := 42; // *
    CHAR_LAZINESS: DWORD := 63; // ?
    CHAR_DOT: DWORD := 46; // .
    CHAR_ESCAPE: DWORD := 92; // \
END_VAR

FuCompilePatternW := FALSE;

IF udiPatternLength = 0 THEN
    RETURN;
END_IF

tempPointer := pwsPattern;

i := 0;
tempMaxStrIndex := udiPatternLength - 1;

WHILE i <= tempMaxStrIndex DO
    IF tempIndex > ParameterList.uiMaxPatternTokens THEN
        EXIT;
    END_IF
    
    IF NOT FuUtf16CharToDword(psInput := (tempPointer + (i * 2)), udiStringLength := (udiPatternLength - (i * 2)), dwCodepoint => tempChar, usiWordLength => tempCharLength) THEN
        RETURN;
    END_IF
    
    IF tempChar = 0 THEN
        EXIT;
    END_IF
    
    IF
        i > tempMaxStrIndex OR_ELSE
        NOT FuUtf16CharToDword(
            psInput := (tempPointer + (i * 2) + (tempCharLength * 2)),
            udiStringLength := (udiPatternLength - (i * 2) - (tempCharLength * 2)),
            dwCodepoint => tempNextChar,
            usiWordLength => tempNextCharLength
        )
    THEN
        tempNextChar := 0;
        tempNextCharLength := 0;
    END_IF
    
    IF tempChar = CHAR_WILDCARD THEN // Wildcard (*)
        typPattern.atTokens[tempIndex].eType := eTokenType.WILDCARD;
        typPattern.atTokens[tempIndex].dwChar := 0; // Use dwChar as modifier to be lazy
    ELSIF
        tempChar = CHAR_LAZINESS AND_THEN
        tempIndex > 0 AND_THEN
        typPattern.atTokens[(tempIndex - 1)].eType = eTokenType.WILDCARD
    THEN // Laziness (?), but only if previously wildcard, otherwise literal
        typPattern.atTokens[(tempIndex - 1)].dwChar := 1;
        
        i := i + tempCharLength;
        CONTINUE;
    ELSIF tempChar = CHAR_DOT THEN // Single char (.)
        typPattern.atTokens[tempIndex].eType := eTokenType.ANYCHAR;
    ELSIF
        tempChar = CHAR_ESCAPE AND_THEN (
            tempNextChar = CHAR_WILDCARD OR_ELSE
            tempNextChar = CHAR_DOT
        )
    THEN // Backslash (escape token for . or *, if followed by . or *)
        typPattern.atTokens[tempIndex].eType := eTokenType.LITERAL;
        typPattern.atTokens[tempIndex].dwChar := tempNextChar;
        i := i + tempNextCharLength;
    ELSE
        typPattern.atTokens[tempIndex].eType := eTokenType.LITERAL;
        typPattern.atTokens[tempIndex].dwChar := tempChar;
        
        IF xCaseInsensitive THEN
            // Calculate for the ISO 8859-1 latin1 alphabet the uppercase or lowercase character number (efficient way)
            IF tempChar >= 65 AND_THEN tempChar <= 90 THEN
                // Uppercase A-Z
                tempNextChar := tempChar + 32;
            ELSIF tempChar >= 97 AND_THEN tempChar <= 122 THEN
                // Lowercase a-z
                tempNextChar := tempChar - 32;
            ELSIF tempChar >= 192 AND_THEN tempChar <= 221 AND_THEN tempChar <> 215 THEN
                // Uppercase ISO 8859-1
                tempNextChar := tempChar + 32;
            ELSIF tempChar >= 224 AND_THEN tempChar <= 253 AND_THEN tempChar <> 247 THEN
                // Lowercase ISO 8859-1
                tempNextChar := tempChar - 32; 
            ELSE
                // If we're not in the ISO 8859-1 latin1 alphabet range, use the UTF-8 function to calculate it
                tempNextChar := FuUnicodeCodepointCaseConvert(tempChar);
            END_IF
        ELSE
            tempNextChar := 0;
        END_IF
        
        typPattern.atTokens[tempIndex].dwAlternativeChar := tempNextChar;
    END_IF
    
    tempIndex := tempIndex + 1;
    typPattern.uiCountTokens := tempIndex;
    
    i := i + tempCharLength;
END_WHILE

FuCompilePatternW := (tempIndex > 0);
typPattern.xCaseInsensitive := xCaseInsensitive;

END_FUNCTION

// 20 Program Organization Units/UTF-16/FuUtf16CharToDword
// Calculates for a UTF-16 character from the given WSTRING the codepoint value as DWORD.
// The return value signifies whether the conversion was successful and the codepoint is valid ("well formed").
{attribute 'qualified_only'}
FUNCTION FuUtf16CharToDword : BOOL
VAR_INPUT
    psInput: POINTER TO WSTRING(2);          // A pointer to the string - for technical reasons this is a WSTRING(2), although any length is supported
    udiStringLength: UDINT;                  // The length of the string (in words (length in bytes/2), not codepoints)
END_VAR
VAR_OUTPUT
    dwCodepoint: DWORD;                      // The codepoint value
    usiWordLength: USINT(0..2);              // Provides the codepoint length in words
END_VAR
{library PRIVATE}
VAR
    tempChar1: WORD;
    tempChar2: WORD;
END_VAR

FuUtf16CharToDword := FALSE;
dwCodepoint := 0;
usiWordLength := 0;

IF udiStringLength = 0 THEN
    RETURN;
END_IF

tempChar1 := psInput^[0];

IF tempChar1 >= 16#D800 AND_THEN tempChar1 <= 16#DBFF THEN
    // Two word character
    IF udiStringLength < 2 THEN
        RETURN;
    END_IF
    
    tempChar2 := psInput^[1];
    
    IF NOT FuValidateUtf16BytesForLength2(tempChar1, tempChar2) THEN
        RETURN;
    END_IF
    
    FuUtf16CharToDword := TRUE;
    dwCodepoint := SHL(TO_DWORD(tempChar1), 10) + TO_DWORD(tempChar2) + TO_DWORD((16#10000 - SHL(16#D800, 10) - 16#DC00));
    usiWordLength := 2;
ELSIF (tempChar1 >= 0 AND_THEN tempChar1 <= 16#D7FF) OR_ELSE (tempChar1 >= 16#E000 AND_THEN tempChar1 <= 16#FFFF) THEN
    // One word character
    
    FuUtf16CharToDword := TRUE;
    dwCodepoint := TO_DWORD(tempChar1);
    usiWordLength := 1;
ELSE
    // Invalid leader word value
    RETURN;
END_IF

END_FUNCTION

// 20 Program Organization Units/UTF-16/FuValidateUtf16BytesForLength2
// Checks whether the UTF-16 byte sequence is "well formed" (valid) for 2 word length.
{attribute 'qualified_only'}
FUNCTION FuValidateUtf16BytesForLength2 : BOOL
VAR_INPUT
    wChar1: WORD;
    wChar2: WORD;
END_VAR

FuValidateUtf16BytesForLength2 := (wChar1 >= 16#D800 AND_THEN wChar1 <= 16#DBFF AND_THEN wChar2 >= 16#DC00 AND_THEN wChar2 <= 16#DFFF);

END_FUNCTION

// 20 Program Organization Units/FuMatchExpressionW
// Matches the given compiled pattern against the subject.
// This is the UTF-16 (WSTRING) version of FuMatchExpression.
{attribute 'qualified_only'}
FUNCTION FuMatchExpressionW : BOOL
VAR_INPUT
    typPattern: typCompiledPatternW;      // The compiled pattern from "FuCompilePatternW"
    pwsSubject: POINTER TO WSTRING(1);    // A pointer to the subject string - for technical reasons this is a WSTRING(1), although any size is supported
    udiLength: UDINT;                     // The length of the subject string (in words (length in bytes/2), not codepoints)
END_VAR
{library PRIVATE}
VAR
    tempPtrStr: POINTER TO WORD;
    tempPtrStrMatching: POINTER TO WORD;
    tempStrIndex: UDINT;
    tempStrIndexMatching: UDINT;
    
    i: UINT;
    j: UINT;
    k: LINT;
    
    tempChar: DWORD;
    tempCharLength: USINT;
    
    tempNextChar: DWORD;
    tempNextCharLength: DWORD;
    
    tempLaziness: BOOL;
    tempHasEndChar: BOOL;
    tempEndChar: DWORD;
    tempEndChar2: DWORD;
    
    tempWildcardSearchStart: LINT;
    tempWildcardSearchEnd: LINT;
    tempWildcardSearchBy: LINT;
    tempWildcardSearchOffset: UDINT;
    tempWildcardSearchSuccess: BOOL;
END_VAR

FuMatchExpressionW := FALSE;

IF typPattern.uiCountTokens = 0 OR_ELSE udiLength = 0 THEN
    RETURN;
END_IF

tempPtrStr := pwsSubject;
tempStrIndex := 0;

WHILE i < typPattern.uiCountTokens DO
    IF tempStrIndex >= udiLength THEN
        // Only if all following tokens are of type WILDCARD, we can allow a match to be positive
        FOR j := i TO (typPattern.uiCountTokens - 1) BY 1 DO
            IF typPattern.atTokens[j].eType <> eTokenType.WILDCARD THEN
                FuMatchExpressionW := FALSE;
                RETURN;
            END_IF
        END_FOR
        
        FuMatchExpressionW := TRUE;
        RETURN;
    END_IF
    
    IF NOT FuUtf16CharToDword(psInput := (tempPtrStr + (tempStrIndex * 2)), udiStringLength := (udiLength - (tempStrIndex * 2)), dwCodepoint => tempChar, usiWordLength => tempCharLength) THEN
        RETURN;
    END_IF
    
    CASE typPattern.atTokens[i].eType OF
        eTokenType.INVALID: // We shouldn't ever get an invalid token inside our token array that isn't behind our count
            RETURN;
        
        eTokenType.LITERAL:
            IF
                tempChar <> typPattern.atTokens[i].dwChar AND_THEN
                (
                    NOT typPattern.xCaseInsensitive OR_ELSE
                    typPattern.atTokens[i].dwAlternativeChar = 0 OR_ELSE
                    tempChar <> typPattern.atTokens[i].dwAlternativeChar
                ) 
            THEN
                RETURN;
            END_IF
            
            tempStrIndex := tempStrIndex + tempCharLength;
        
        eTokenType.ANYCHAR:
            tempStrIndex := tempStrIndex + tempCharLength;
        
        eTokenType.WILDCARD:
            tempLaziness := (typPattern.atTokens[i].dwChar = 1);
            tempHasEndChar := FALSE;
            
            FOR j := i + 1 TO (typPattern.uiCountTokens - 1) BY 1 DO
                IF typPattern.atTokens[j].eType = eTokenType.LITERAL THEN
                    tempHasEndChar := TRUE;
                    tempEndChar := typPattern.atTokens[j].dwChar;
                    tempEndChar2 := typPattern.atTokens[j].dwAlternativeChar;
                    EXIT;
                END_IF
            END_FOR
            
            // If we don't have any characters to match on at the end of the pattern, we match immediately
            IF NOT tempHasEndChar THEN
                FuMatchExpressionW := TRUE;
                RETURN;
            END_IF
            
            IF tempLaziness THEN
                // Advance token pointer once more because the next token is the laziness token we already used
                i := i + 1;
                
                // If the wildcard is lazy, search from front to back
                tempWildcardSearchStart := TO_LINT(tempStrIndex);
                tempWildcardSearchEnd := TO_LINT(udiLength);
                tempWildcardSearchBy := 1;
            ELSE
                // If the wildcard is NOT lazy, search from back to front (greedy!)
                tempWildcardSearchStart := TO_LINT(udiLength);
                tempWildcardSearchEnd := TO_LINT(tempStrIndex);
                tempWildcardSearchBy := -1;
            END_IF
            
            tempWildcardSearchSuccess := FALSE;
            tempWildcardSearchOffset := 0;
            
            FOR k := tempWildcardSearchStart TO tempWildcardSearchEnd BY tempWildcardSearchBy DO
                IF
                    FuUtf16CharToDword(
                        psInput := (tempPtrStr + LINT_TO___XWORD(k)),
                        udiStringLength := (udiLength - tempWildcardSearchOffset),
                        dwCodepoint => tempNextChar,
                        usiWordLength => tempNextCharLength
                    )
                THEN
                    tempWildcardSearchOffset := tempWildcardSearchOffset + tempNextCharLength;
                    
                    IF
                        tempNextChar = tempEndChar OR_ELSE
                        (typPattern.xCaseInsensitive AND_THEN tempEndChar2 <> 0 AND_THEN tempNextChar = tempEndChar2)
                    THEN
                        tempWildcardSearchSuccess := TRUE;
                        tempStrIndex := TO_UDINT(k);
                        EXIT;
                    END_IF
                ELSE
                    tempWildcardSearchOffset := tempWildcardSearchOffset + 1;
                END_IF
            END_FOR
            
            IF NOT tempWildcardSearchSuccess THEN
                RETURN;
            END_IF
    END_CASE
    
    i := i + 1;
END_WHILE

FuMatchExpressionW := (tempStrIndex >= udiLength);

END_FUNCTION

// 20 Program Organization Units/FuCompilePatternW2
// Same as FuCompilePatternW, except it doesn't take a pointer and has a fixed length.
{attribute 'qualified_only'}
FUNCTION FuCompilePatternW2 : BOOL
VAR_INPUT
    wsPattern: WSTRING(255);              // The pattern string to compile
    xCaseInsensitive: BOOL := FALSE;      // Whether the pattern is case insensitive
END_VAR
VAR_OUTPUT
    typPattern: typCompiledPatternW;      // The compiled pattern, for "FuMatchExpressionW"
END_VAR

FuCompilePatternW2 := FuCompilePatternW(ADR(wsPattern), TO_UDINT(Stu.StrLenW(ADR(wsPattern))), xCaseInsensitive, typPattern => typPattern);

END_FUNCTION
